// TIA Portal V20 export
DATA_BLOCK "DB_AsiSetpoint"   // DB28
// stored: Access Published, MemoryReserve 100, Namespace LineC1
   VAR
      Line : Struct
         C1 : Struct
            DirChange : Struct
               Conveyor : Array[_.minC1.._.maxC1] of Bool;
            END_STRUCT;
            Speed : Struct
               Conveyor : Array[_.minC1.._.maxC1] of Bool;
            END_STRUCT;
         END_STRUCT;
      END_STRUCT;
   END_VAR
BEGIN
END_DATA_BLOCK
